FUNCTION_BLOCK COMMCHANNEL (* Service Interface Function Block Type *)
  (* Standard: 61499-2 *)
  (* Version 0.0, 9/14/2008, Horst Mayer, nxtControl GmbH, template *)
  PACKAGE IEC61499;
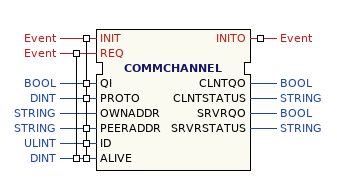
  EVENT_INPUT
    INIT WITH QI, PROTO, PEERADDR, ID, ALIVE;
    REQ WITH ALIVE;
  END_EVENT
  EVENT_OUTPUT
    INITO WITH QO, STATUS;
  END_EVENT
  VAR_INPUT
    QI : BOOL;
    PROTO : DINT;
    OWNADDR : STRING;
    PEERADDR : STRING;
    ID : ULINT;
    ALIVE : DINT;
  END_VAR
  VAR_OUTPUT
    CLNTQO : BOOL; (* Event Output Qualifier *)
    CLNTSTATUS : STRING; (* Service Status *)
    SRVRQO : BOOL; (* Event Output Qualifier *)
    SRVRSTATUS : STRING; (* Service Status *)
  END_VAR
END_FUNCTION_BLOCK
